# EPICS substitutions: evrSupport/Db/ioc/IOC-IN20-LS11trig.substitutions
# Trigger records
#
# refer to Sharepoint document: Controls | Timing | timingTriggers.xls
#
# Must also have pattern records
# Note: WID, DES, TEC are in terms of nSec and are unique per device
#
file evrDevTrig.db {
#      Device	      , Description   , EVR  ,  width ,desired  , EC delay   , EVR  , EVR,  IOC          , slope
#			                            Trigger       wrt TREF   wrt fiducial loca   unit                 1/119Mhz
  pattern { DEV       ,  DESC         , T    ,  WID   , DES     , TEC       , LOCA , UNIT, IOC          , ESLO
                      ,  PREC         , EGU  ,  DRVL  , DRVH    , EVG       , OTP}
	  { AFG:IN20:LS11: ,  "Horiz Drive", 0    ,  100   , 10      , TS4_10_  , IN20 , LS11, IOC:IN20:LS11, 8.40336692324359
                      ,  1            ,"nSec", -2.8E06, 2.8E06  , IN20:EV01 , OTP0}
	  { CAMR:IN20:LS11:, "Vert Drive"  , 1    ,  100   , 10      , TS4_10_  , IN20 , LS11, IOC:IN20:LS11, 8.40336692324359
                      ,  1            ,"nSec", -2.8E06, 2.8E06  , IN20:EV01 , OTP1}
	  { ADC:IN20:LS11: , "ADC 1"       , 2    ,  100   , 10      , TS4_10_  , IN20 , LS11, IOC:IN20:LS11, 8.40336692324359
                      ,  1            ,"nSec", -2.8E06, 2.8E06  , IN20:EV01 , OTP2}
}
